FUNCTION_BLOCK FB_LimSwStatus IMPLEMENTS I_LimSwStatus
VAR_INPUT
END_VAR
VAR_OUTPUT
END_VAR
VAR
    {attribute 'hide'}
    iMotionLogger	: I_MotionLogger;

    (* Hardware *)
   // NC Forward Limit Switch: TRUE if ok to move
    bLimitForwardEnable AT %I*: BOOL;
    // NC Backward Limit Switch: TRUE if ok to move
    bLimitBackwardEnable AT %I*: BOOL;
    // NO Home Switch: TRUE if at home
    bHome AT %I*: BOOL;

    {attribute 'hide'}
    bLimHit : BOOL;
    bMoveBackwardEnabled : BOOL;
    bMoveForwardEnabled : BOOL;
    {attribute 'hide'}
    ftForwardEnabled : F_TRIG;
    {attribute 'hide'}
    ftBackwardEnabled : F_TRIG;
    {attribute 'hide'}
    rtUserExec : R_TRIG;
    {attribute 'hide'}
    rtReset : R_TRIG;
    {attribute 'hide'}
    bLimHitIdling : BOOL;
    {attribute 'hide'}
    bLimHitMoving : BOOL;
    {attribute 'hide'}
    bWarning: BOOL;
    {attribute 'hide'}
    sMessage: T_MAXSTRING;
    {attribute 'hide'}
    bNewMoveReq : BOOL;
    {attribute 'hide'}
    bEnable	: BOOL;
    {attribute 'hide'}
    bReset : BOOL;
    {attribute 'hide'}
    bPositiveDirection : BOOL;
    {attribute 'hide'}
    bNegativeDirection : BOOL;
    {attribute 'hide'}
    bHomeBusy : BOOL;
    bLimForward : BOOL;
    bLimBackward: BOOL;
    bLimHome: BOOL;
END_VAR

// Read Limits status and update shared space
bMoveBackwardEnabled := bLimitBackwardEnable;
bMoveForwardEnabled := bLimitForwardEnable;

// Todo: axis idling, critical limit disable faillure
// clear previous warning and limit hit events with each new request
// wait for global reset event to complete
rtReset(CLK:=bReset);
rtUserExec (CLK:=bNewMoveReq);
ftForwardEnabled(CLK:=bMoveForwardEnabled);
ftBackwardEnabled (CLK:=bMoveBackwardEnabled);

IF NOT THIS^.bHomeBusy AND ((ftForwardEnabled.Q AND THIS^.bPositiveDirection)
        OR (ftBackwardEnabled.Q AND THIS^.bNegativeDirection))THEN
    // Not an error, just a warning
    IF NOT bMoveForwardEnabled THEN
            THIS^.sMessage:='Cannot move past Positive limit.';
    ELSIF NOT bMoveBackwardEnabled THEN
            THIS^.sMessage:='Cannot move past Negative limit.';
    END_IF
    THIS^.bWarning:=TRUE;
    THIS^.bLimHit := TRUE;
    THIS^.bLimHitMoving:=TRUE;
ELSIF rtUserExec.Q OR rtReset.Q THEN
    THIS^.bLimHit := FALSE;
    THIS^.bLimHitMoving := bLimHit;
    THIS^.bLimHitIdling := bLimHit;
    THIS^.sMessage := '';
    THIS^.bWarning := FALSE;
END_IF

METHOD AxisStatus
VAR_INPUT
    HomeBusy: BOOL;
    PositiveDirection : BOOL;
    NegativeDirection : BOOL;
END_VAR
bHomeBusy :=HomeBusy;
bPositiveDirection :=PositiveDirection;
bNegativeDirection :=NegativeDirection;
END_METHOD

METHOD DriveCommands
VAR_INPUT
    Enable	: BOOL;
    NewMoveReq	: BOOL;
    Reset	: BOOL;
END_VAR
THIS^.bEnable := Enable;
THIS^.bReset := Reset;
THIS^.bNewMoveReq := NewMoveReq ;
END_METHOD

//FB_Init is always available implicitly and it is used primarily for initialization.
//The return value is not evaluated. For a specific influence, you can also declare the
//methods explicitly and provide additional code there with the standard initialization
//code. You can evaluate the return value.
METHOD FB_Init: BOOL
VAR_INPUT
    bInitRetains: BOOL; // TRUE: the retain variables are initialized (reset warm / reset cold)
    bInCopyCode: BOOL;  // TRUE: the instance will be copied to the copy code afterward (online change)
    iMotionLogger	: I_MotionLogger;
END_VAR
END_METHOD

{warning 'add property implementation'}
PROPERTY LimBackward : BOOL
GET
LimBackward := bLimitBackwardEnable;
END_GET
END_PROPERTY

{warning 'add property implementation'}
PROPERTY LimForward : BOOL
GET
LimForward := bLimitForwardEnable;
END_GET
END_PROPERTY

PROPERTY LimHit : BOOL
GET
LimHit := bLimHit;
END_GET
END_PROPERTY

{warning 'Add property implementation'}
PROPERTY LimHitIdling : BOOL
GET
END_GET
END_PROPERTY

{warning 'Add property implementation'}
PROPERTY LimHitMoving : BOOL
GET
END_GET
END_PROPERTY

{warning 'add property implementation'}
PROPERTY LimHome : BOOL
GET
LimHome := bHome;
END_GET
END_PROPERTY

{warning 'Add property implementation'}
PROPERTY Message : T_MAXSTRING
GET
Message := sMessage;
END_GET
END_PROPERTY

PROPERTY MoveBackwardEnabled : BOOL
GET
MoveBackwardEnabled := bMoveBackwardEnabled;
END_GET
END_PROPERTY

PROPERTY MoveForwardEnabled : BOOL
GET
MoveForwardEnabled := bMoveForwardEnabled;
END_GET
END_PROPERTY

PROPERTY Warning : BOOL
GET
 Warning := bWarning;
END_GET
END_PROPERTY

END_FUNCTION_BLOCK

(* stored: Version 1.1.0.1
   POU FB_LimSwStatus: Id {322e8186-deb9-4a53-b303-d1d3662306db}, SpecialFunc None
   Method AxisStatus: Id {a1a77b92-9069-4c95-afb6-6e44858fa0e1}
   Method DriveCommands: Id {b140fe49-9bf2-4392-9913-139634acc355}
   Method FB_Init: Id {e9d4b1d6-7e2a-40e5-abfc-b6d7871092e6}
   Property LimBackward: Id {aa63489c-6e6a-4b3c-98b7-5f6f7e3fb754}
   Get Get: Id {134e6218-84e4-4ed6-bfc7-d7acf7d3e2e8}
   Property LimForward: Id {2df92432-ddf8-46fa-9ca0-e9671149f768}
   Get Get: Id {c1785027-3e2e-4947-b69b-9e7918a456b0}
   Property LimHit: Id {f510c7ce-a1d2-4aed-84bc-03f1d019d2f4}
   Get Get: Id {1e5d3be5-c543-46b8-afd6-4d69c846bbb6}
   Property LimHitIdling: Id {e2383759-743f-482f-a670-ac8df1ae3fbf}
   Get Get: Id {4bef7835-b757-492b-9d0a-0abd3adc4ac8}
   Property LimHitMoving: Id {6aaf6510-ab50-4511-8a06-874853bf780d}
   Get Get: Id {b942862e-5cc6-495e-8cc1-f1909d9ecaa8}
   Property LimHome: Id {bb43c80f-c8b0-49cb-8388-6e64188fca33}
   Get Get: Id {fb83aff6-4f66-438e-8ea7-ee58a5c4ea24}
   Property Message: Id {b08158f2-a8bc-4fe9-8e03-fb8deb3f9f62}
   Get Get: Id {6db79a56-c326-4a16-8442-f3020ce04421}
   Property MoveBackwardEnabled: Id {89adc283-9c17-45ca-8f36-46140fc4dc4c}
   Get Get: Id {3db33672-1b0d-4c45-b399-57143d800f06}
   Property MoveForwardEnabled: Id {5cf35d17-2e51-4927-83dd-9d0c0496a7d4}
   Get Get: Id {157158b2-9f48-4b44-a9b9-77a750c8b408}
   Property Warning: Id {c7ddb3f1-3a2c-446a-8003-00c9756105d6}
   Get Get: Id {1f972676-2f12-4b3f-adb4-9a49850d0be5} *)
